TYPE stCorkMachine EXTENDS stPimMachineData :
STRUCT
	
END_STRUCT
END_TYPE

(* stored: Version 1.1.0.1, ProductVersion 3.1.4024.13
   DUT stCorkMachine: Id {c2d04ca5-9436-4a4b-ba26-27f537b9c496} *)
